// TIA Portal V18 export
// export: Created 2026-04-18T00:00:00Z, ExportSetting WithDefaults
FUNCTION "FC_Init_Default_Recipe_PLC1" : Void   // FC50, LAD
{ S7_Optimized_Access := 'TRUE' }
VERSION : 0.1
// stored: AutoNumber true, IsIECCheckEnabled false
BEGIN

REGION Network 1: Kích hoạt nạp recipe mặc định lần đầu scan PLC1
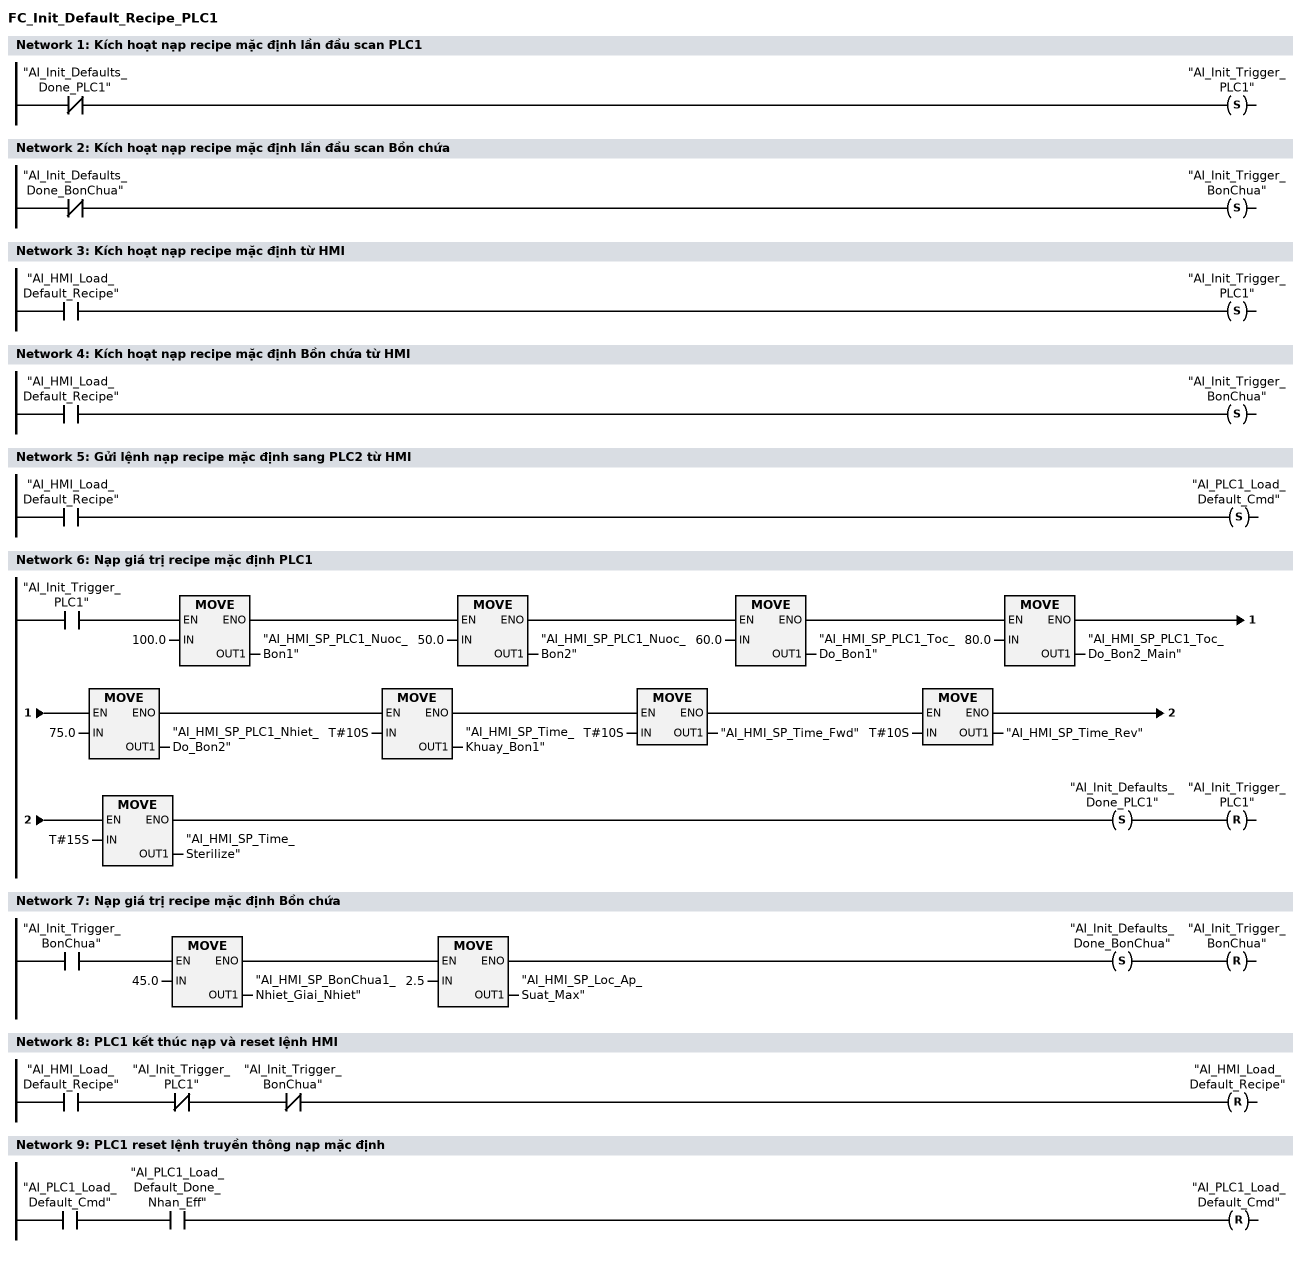
   RUNG wire#powerrail
      I_Contact( "AI_Init_Defaults_Done_PLC1" )
      S_Coil( "AI_Init_Trigger_PLC1" )
   END_RUNG
   // the same network as SCL:
   IF NOT "AI_Init_Defaults_Done_PLC1" THEN "AI_Init_Trigger_PLC1" := TRUE; END_IF;
END_REGION

REGION Network 2: Kích hoạt nạp recipe mặc định lần đầu scan Bồn chứa
   RUNG wire#powerrail
      I_Contact( "AI_Init_Defaults_Done_BonChua" )
      S_Coil( "AI_Init_Trigger_BonChua" )
   END_RUNG
   // the same network as SCL:
   IF NOT "AI_Init_Defaults_Done_BonChua" THEN "AI_Init_Trigger_BonChua" := TRUE; END_IF;
END_REGION

REGION Network 3: Kích hoạt nạp recipe mặc định từ HMI
   RUNG wire#powerrail
      Contact( "AI_HMI_Load_Default_Recipe" )
      S_Coil( "AI_Init_Trigger_PLC1" )
   END_RUNG
   // the same network as SCL:
   IF "AI_HMI_Load_Default_Recipe" THEN "AI_Init_Trigger_PLC1" := TRUE; END_IF;
END_REGION

REGION Network 4: Kích hoạt nạp recipe mặc định Bồn chứa từ HMI
   RUNG wire#powerrail
      Contact( "AI_HMI_Load_Default_Recipe" )
      S_Coil( "AI_Init_Trigger_BonChua" )
   END_RUNG
   // the same network as SCL:
   IF "AI_HMI_Load_Default_Recipe" THEN "AI_Init_Trigger_BonChua" := TRUE; END_IF;
END_REGION

REGION Network 5: Gửi lệnh nạp recipe mặc định sang PLC2 từ HMI
   RUNG wire#powerrail
      Contact( "AI_HMI_Load_Default_Recipe" )
      S_Coil( "AI_PLC1_Load_Default_Cmd" )
   END_RUNG
   // the same network as SCL:
   IF "AI_HMI_Load_Default_Recipe" THEN "AI_PLC1_Load_Default_Cmd" := TRUE; END_IF;
END_REGION

REGION Network 6: Nạp giá trị recipe mặc định PLC1
   RUNG wire#powerrail
      Contact( "AI_Init_Trigger_PLC1" )
      { S7_GenerateENO := "TRUE" } Move(in := 100.0, out1 => "AI_HMI_SP_PLC1_Nuoc_Bon1")
      { S7_GenerateENO := "TRUE" } Move(in := 50.0, out1 => "AI_HMI_SP_PLC1_Nuoc_Bon2")
      { S7_GenerateENO := "TRUE" } Move(in := 60.0, out1 => "AI_HMI_SP_PLC1_Toc_Do_Bon1")
      { S7_GenerateENO := "TRUE" } Move(in := 80.0, out1 => "AI_HMI_SP_PLC1_Toc_Do_Bon2_Main")
      { S7_GenerateENO := "TRUE" } Move(in := 75.0, out1 => "AI_HMI_SP_PLC1_Nhiet_Do_Bon2")
      { S7_GenerateENO := "TRUE" } Move(in := T#10S, out1 => "AI_HMI_SP_Time_Khuay_Bon1")
      { S7_GenerateENO := "TRUE" } Move(in := T#10S, out1 => "AI_HMI_SP_Time_Fwd")
      { S7_GenerateENO := "TRUE" } Move(in := T#10S, out1 => "AI_HMI_SP_Time_Rev")
      { S7_GenerateENO := "TRUE" } Move(in := T#15S, out1 => "AI_HMI_SP_Time_Sterilize")
      S_Coil( "AI_Init_Defaults_Done_PLC1" )
      R_Coil( "AI_Init_Trigger_PLC1" )
   END_RUNG
   // the same network as SCL:
   // ENO of a box is taken as its EN; it also drops when the box reports an error
   IF "AI_Init_Trigger_PLC1" THEN
       "AI_HMI_SP_PLC1_Nuoc_Bon1" := 100.0;
       "AI_HMI_SP_PLC1_Nuoc_Bon2" := 50.0;
       "AI_HMI_SP_PLC1_Toc_Do_Bon1" := 60.0;
       "AI_HMI_SP_PLC1_Toc_Do_Bon2_Main" := 80.0;
       "AI_HMI_SP_PLC1_Nhiet_Do_Bon2" := 75.0;
       "AI_HMI_SP_Time_Khuay_Bon1" := T#10S;
       "AI_HMI_SP_Time_Fwd" := T#10S;
       "AI_HMI_SP_Time_Rev" := T#10S;
       "AI_HMI_SP_Time_Sterilize" := T#15S;
       "AI_Init_Defaults_Done_PLC1" := TRUE;
       "AI_Init_Trigger_PLC1" := FALSE;
   END_IF;
END_REGION

REGION Network 7: Nạp giá trị recipe mặc định Bồn chứa
   RUNG wire#powerrail
      Contact( "AI_Init_Trigger_BonChua" )
      { S7_GenerateENO := "TRUE" } Move(in := 45.0, out1 => "AI_HMI_SP_BonChua1_Nhiet_Giai_Nhiet")
      { S7_GenerateENO := "TRUE" } Move(in := 2.5, out1 => "AI_HMI_SP_Loc_Ap_Suat_Max")
      S_Coil( "AI_Init_Defaults_Done_BonChua" )
      R_Coil( "AI_Init_Trigger_BonChua" )
   END_RUNG
   // the same network as SCL:
   // ENO of a box is taken as its EN; it also drops when the box reports an error
   IF "AI_Init_Trigger_BonChua" THEN
       "AI_HMI_SP_BonChua1_Nhiet_Giai_Nhiet" := 45.0;
       "AI_HMI_SP_Loc_Ap_Suat_Max" := 2.5;
       "AI_Init_Defaults_Done_BonChua" := TRUE;
       "AI_Init_Trigger_BonChua" := FALSE;
   END_IF;
END_REGION

REGION Network 8: PLC1 kết thúc nạp và reset lệnh HMI
   RUNG wire#powerrail
      Contact( "AI_HMI_Load_Default_Recipe" )
      I_Contact( "AI_Init_Trigger_PLC1" )
      I_Contact( "AI_Init_Trigger_BonChua" )
      R_Coil( "AI_HMI_Load_Default_Recipe" )
   END_RUNG
   // the same network as SCL:
   IF "AI_HMI_Load_Default_Recipe" AND NOT "AI_Init_Trigger_PLC1" AND NOT "AI_Init_Trigger_BonChua" THEN
       "AI_HMI_Load_Default_Recipe" := FALSE;
   END_IF;
END_REGION

REGION Network 9: PLC1 reset lệnh truyền thông nạp mặc định
   RUNG wire#powerrail
      Contact( "AI_PLC1_Load_Default_Cmd" )
      Contact( "AI_PLC1_Load_Default_Done_Nhan_Eff" )
      R_Coil( "AI_PLC1_Load_Default_Cmd" )
   END_RUNG
   // the same network as SCL:
   IF "AI_PLC1_Load_Default_Cmd" AND "AI_PLC1_Load_Default_Done_Nhan_Eff" THEN
       "AI_PLC1_Load_Default_Cmd" := FALSE;
   END_IF;
END_REGION
END_FUNCTION
